FUNCTION_BLOCK Server (* Template for a Basic Function Block Type *)
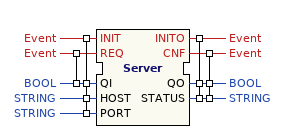
  EVENT_INPUT
    INIT WITH QI, HOST, PORT; (* Initialization Request *)
    REQ WITH QI; (* Normal Execution Request *)
  END_EVENT
  EVENT_OUTPUT
    INITO WITH QO, STATUS; (* Initialization Confirm *)
    CNF WITH QO, STATUS; (* Execution Confirmation *)
  END_EVENT
  VAR_INPUT
    QI : BOOL; (* Input event qualifier *)
    HOST : STRING;
    PORT : STRING;
  END_VAR
  VAR_OUTPUT
    QO : BOOL; (* Output event qualifier *)
    STATUS : STRING;
  END_VAR
END_FUNCTION_BLOCK
